PROGRAM MAIN
VAR
END_VAR

END_PROGRAM

(* stored: Version 1.1.0.1
   POU MAIN: Id {8a779814-4d9f-40e5-ab78-160e9e5cefe7} *)
